FUNCTION_BLOCK FB_LiftCylinderBosch EXTENDS FB_Cylinder
VAR
(*----------------------------------------------------------------------------------------------*)
	sensorMID		AT %I*		: BOOL;
(*----------------------------------------------------------------------------------------------*)
	_inMID						: BOOL;
	_newStateInterlockMID		: BOOL;
	_newStateInterlockMsgMID	: STRING(255);
	_interlockMID				: BOOL;
	_interlockMessageMID		: STRING(255);
	_sensorTagMID				: STRING;
	_notUsedSensorMID			: BOOL;
	_delayTimeAfterReachedMID	: TIME;
	_timerInMID					: Tc2_Standard.TON;	
(*----------------------------------------------------------------------------------------------*)
END_VAR

METHOD INTERNAL _handleInterlocks
VAR_INPUT
END_VAR
(*----------------------------------------------------------------------------------------------*)
_interlockHP:= _newStateInterlockHP;
_interlockMessageHP:= _newStateInterlockMsgHP;
_newStateInterlockHP:= FALSE;
_newStateInterlockMsgHP:= '';
(*----------------------------------------------------------------------------------------------*)
_interlockMID:= _newStateInterlockMID;
_interlockMessageMID:= _newStateInterlockMsgMID;
_newStateInterlockMID:= FALSE;
_newStateInterlockMsgMID:= '';
(*----------------------------------------------------------------------------------------------*)
_interlockWP:= _newStateInterlockWP;
_interlockMessageWP:= _newStateInterlockMsgWP;
_newStateInterlockWP:= FALSE;
_newStateInterlockMsgWP:= '';
(*----------------------------------------------------------------------------------------------*)
END_METHOD

METHOD INTERNAL _handlePositionStatus
VAR_INPUT
END_VAR
(*----------------------------------------------------------------------------------------------*)
_timerInHP(
	IN	:= valveHP AND (_notUsedSensorHP OR sensorHP) AND (NOT sensorWP OR NOT _Config.monitorSensorsOverlap),
	PT	:= _Config.delayTimeAfterReachedHP,
	Q	=> _inHP);
(*----------------------------------------------------------------------------------------------*)
_timerInMID(
	IN	:= NOT valveHP AND NOT valveWP AND (_notUsedSensorMID OR sensorMID) AND (NOT sensorHP OR NOT _Config.monitorSensorsOverlap) AND (NOT sensorWP OR NOT _Config.monitorSensorsOverlap),
	PT	:= _delayTimeAfterReachedMID,
	Q	=> _inMID);
(*----------------------------------------------------------------------------------------------*)
_timerInWP(
	IN	:= valveWP AND (_notUsedSensorWP OR sensorWP) AND (NOT sensorHP OR NOT _Config.monitorSensorsOverlap),
	PT	:= _Config.delayTimeAfterReachedWP,
	Q	=> _inWP);
(*----------------------------------------------------------------------------------------------*)
_timerTimeout(
	IN:= (_calledMethod <> ''),
	PT:= _Config.movementTimeout);
(*----------------------------------------------------------------------------------------------*)
_timerSensorsOverlap(
	IN:= _Config.monitorSensorsOverlap AND sensorHP AND sensorWP,
	PT:= _Config.sensorsOverlapTimeout);
(*----------------------------------------------------------------------------------------------*)
END_METHOD

METHOD PROTECTED _onInit
VAR_INST
	_isInit				: BOOL;
END_VAR
(*----------------------------------------------------------------------------------------------*)
IF _isInit THEN RETURN; END_IF
(*----------------------------------------------------------------------------------------------*)
IF (_sensorTagHP = '') THEN
	_notUsedSensorHP:= TRUE;
END_IF
(*----------------------------------------------------------------------------------------------*)
IF (_sensorTagMID = '') THEN
	_notUsedSensorMID:= TRUE;
END_IF
(*----------------------------------------------------------------------------------------------*)
IF (_sensorTagWP = '') THEN
	_notUsedSensorWP:= TRUE;
END_IF
(*----------------------------------------------------------------------------------------------*)
_isInit:= TRUE;
(*----------------------------------------------------------------------------------------------*)
END_METHOD

METHOD addInterlockMID
VAR_INPUT
	condition		: BOOL;
	message			: STRING(255);
END_VAR
IF condition THEN
	_newStateInterlockMID:= TRUE;
	_newStateInterlockMsgMID:= message;
END_IF
END_METHOD

PROPERTY delayTimeAfterReachedMID : TIME
GET
delayTimeAfterReachedMID:= _delayTimeAfterReachedMID;
END_GET
SET
_delayTimeAfterReachedMID:= delayTimeAfterReachedMID;
END_SET
END_PROPERTY

METHOD FB_init : BOOL
VAR_INPUT
	bInitRetains 	: BOOL; 	// if TRUE, the retain variables are initialized (warm start / cold start)
	bInCopyCode 	: BOOL;  	// if TRUE, the instance afterwards gets moved into the copy code (online change)
	name			: STRING;	// identifier for HMI display and logging, example Clipping cylinder
	tag				: STRING;	// el. schematic tag for device, example C1, 10MM1, Z1, etc.
	sensorTagHP		: STRING;	// el. schematic tag for home position sensor input, leave empty '' if no HP sensor attached
	sensorTagWP		: STRING;	// el. schematic tag for work position sensor input, leave empty '' if no WP sensor attached
	sensorTagMID	: STRING;	// el. schematic tag for mid position sensor input, leave empty '' if no MID sensor attached
END_VAR
THIS^._sensorTagMID:= sensorTagMID;
END_METHOD

PROPERTY PUBLIC inMID : BOOL
GET
inMID:= _inMID;
END_GET
END_PROPERTY

METHOD PUBLIC moveToMID
VAR_INPUT
	Response		: REFERENCE TO TcNexa_Components_TcProcess.FB_MethodResponse;
END_VAR
_methodState:= _methodHeader(methodName:= 'move to MID');

IF _methodState.execute THEN
	IF NOT _interlockMID THEN
		valveHP:= FALSE;
		valveWP:= FALSE;		
		(* Error - all sensors active *)
		IF _timerSensorsOverlap.Q THEN
			_InternalResponse.setFail(message:= _getErrorMessage(), description:= 'All sensors active');
		(* Error movement - end position not reached *)		
		ELSIF _timerTimeout.Q THEN
			_InternalResponse.setFail(message:= _getErrorMessage(), description:= _getErrorMsgPositionNotReached(_sensorTagMID));
		(* Succes - end position reached *)
		ELSIF _timerInMID.Q THEN
			_InternalResponse.setPass();
		END_IF	
	ELSE
		_InternalResponse.setFail(message:= _getMsgInterlocked(), description:= _interlockMessageMID);
	END_IF
END_IF

_methodFooter(Response:= Response);
END_METHOD

END_FUNCTION_BLOCK

(* stored: Version 1.1.0.1, ProductVersion 3.1.4026.17
   POU FB_LiftCylinderBosch: Id {cd998b1a-dcf2-035a-166d-956628307c66}, SpecialFunc None
   Folder Internal: Id {2b6daefa-650d-0f24-2fc8-559a700c9078}
   Folder Property: Id {05a26ced-c226-0e15-0293-3d5097c6c6e0}
   Method _handleInterlocks: Id {7c1316e0-e86d-0ad2-0183-4f37e18405db}
   Method _handlePositionStatus: Id {8cc11a2f-bdd6-0f92-0cf6-98319b8dd1b7}
   Method _onInit: Id {c912801e-c395-0264-30af-e08bac4ddd9d}
   Method addInterlockMID: Id {c9b7d522-be9a-0489-2d2f-2afa8918693e}
   Property delayTimeAfterReachedMID: Id {129f627b-7b47-0256-18bc-3560478d814c}
   Get Get: Id {1221ac0f-82db-0bb7-01a2-2ff08d13bd52}
   Set Set: Id {1838641b-a781-0aed-1ce4-4df53a688357}
   Method FB_init: Id {b47e510c-c13e-0423-02cd-91f086977516}
   Property inMID: Id {5abbd232-88f0-05ff-286d-7981a8a11b57}
   Get Get: Id {e449f219-d992-03a9-2cc3-7002d2a5e35a}
   Method moveToMID: Id {68cb3ece-96b9-0619-21e0-15d367a296a0} *)
